{attribute 'GeneratedUsingTerminal: EL3255-0000-0016'}
{attribute addProperty BoxType "EL3255-0000-0016"}
{attribute addProperty Id "RTD_Standard_Channel_1AT %I*RTD_Standard_Channel_A8DF64E310RTD_Standard_Channel_2AT %I*RTD_Standard_Channel_A8DF64E310RTD_Standard_Channel_3AT %I*RTD_Standard_Channel_A8DF64E310RTD_Standard_Channel_4AT %I*RTD_Standard_Channel_A8DF64E310RTD_Standard_Channel_5AT %I*RTD_Standard_Channel_A8DF64E310WcStateAT %I*WcState_9091E0EB2InfoDataAT %I*InfoData_94A18F5E2"}
{attribute addProperty CRC "829931341"}
{attribute addProperty Size "54"}
TYPE EL3255_3177BF4D EXTENDS EtcSlaveTerminalBase_947E5A46 :
STRUCT
	{attribute addProperty Name "RTD_Standard_Channel_1"}
	RTD_Standard_Channel_1 : RTD_Standard_Channel_A8DF64E3;
	{attribute addProperty Name "RTD_Standard_Channel_2"}
	RTD_Standard_Channel_2 : RTD_Standard_Channel_A8DF64E3;
	{attribute addProperty Name "RTD_Standard_Channel_3"}
	RTD_Standard_Channel_3 : RTD_Standard_Channel_A8DF64E3;
	{attribute addProperty Name "RTD_Standard_Channel_4"}
	RTD_Standard_Channel_4 : RTD_Standard_Channel_A8DF64E3;
	{attribute addProperty Name "RTD_Standard_Channel_5"}
	RTD_Standard_Channel_5 : RTD_Standard_Channel_A8DF64E3;
	{attribute addProperty Name "WcState"}
	WcState : WcState_9091E0EB;
	{attribute addProperty Name "InfoData"}
	InfoData : InfoData_94A18F5E;
END_STRUCT
END_TYPE

(* stored: Version 1.2.0.0, ProductVersion 3.1.4024.9
   DUT EL3255_3177BF4D: Id {a09a8a6a-9479-4391-9f37-5f08acc1ca5c} *)
